(* Passes one WORD read across the arbiter bridge. The caller links the raw PDO value and derives
   bridge health elsewhere (e.g. FB_SubSysToArbiter_IO.bBridgeOk) and passes both in each cycle; this
   FB owns no hardware links. Integers have no invalid-bit-pattern to sanitize, so it holds the last
   trusted value while the bridge is down. Error carries only the test override; fault on bad comms
   via the bridge FB's bBridgeConfirmedBad in the caller. *)
FUNCTION_BLOCK FB_FallibleWordFromEtherCAT
IMPLEMENTS I_FallibleWord
VAR_INPUT
    i_bBridgeOk : BOOL;
    i_nValue : WORD;
END_VAR
VAR_OUTPUT
    {attribute 'pytmc' := '
        pv: Value
        io: i
    '}
    nValue : WORD;
END_VAR
VAR
    nLastValidValue : WORD;
    bOverride : BOOL;
    bOverrideError : BOOL;
    nOverrideValue : WORD;
END_VAR


IF i_bBridgeOk THEN
    nLastValidValue := i_nValue;
END_IF

nValue := SEL(bOverride, SEL(i_bBridgeOk, nLastValidValue, i_nValue), nOverrideValue);


PROPERTY Error : BOOL
GET

Error := SEL(bOverride, FALSE, bOverrideError);
END_GET
END_PROPERTY


PROPERTY Value : WORD
GET

Value := THIS^.nValue;
END_GET
END_PROPERTY

END_FUNCTION_BLOCK

(* stored: Version 1.1.0.1
   POU FB_FallibleWordFromEtherCAT: Id {a1b2c3d4-0101-4001-8001-000000000101}, SpecialFunc None
   Property Error: Id {a1b2c3d4-0101-4001-8001-000000000102}
   Get Get: Id {a1b2c3d4-0101-4001-8001-000000000103}
   Property Value: Id {a1b2c3d4-0101-4001-8001-000000000104}
   Get Get: Id {a1b2c3d4-0101-4001-8001-000000000105} *)
